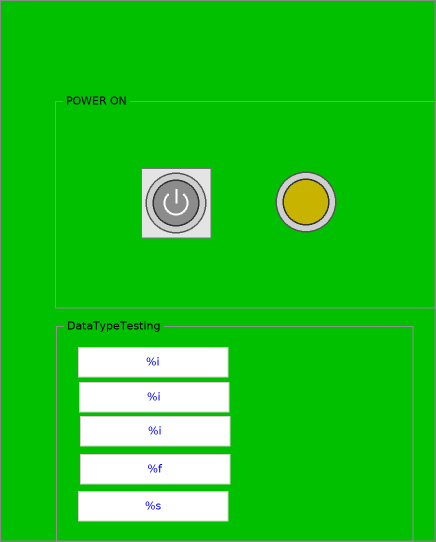
VISUALIZATION HMI  // 436x542
    GroupBox (55,93 381x215), "POWER ON"
        Lamp1 (216,74 70x70), variable: MAIN.bEnable, style: Lamp-Lamp1-Yellow
        PowerSwitch (86,75 70x70), variable: MAIN.bStart, behaviour: TOGGLE, style: Switch-PowerSwitch-Gray
    GroupBox (56,318 357x224), "DataTypeTesting"
        Textfield (22,29 150x30), "%i", text variable: MAIN.bEnable
        Textfield (23,64 150x30), "%i", text variable: MAIN.nINT
        Textfield (22,173 150x30), "%s", text variable: MAIN.sPowerStatus
            OnMouseDown: write the text variable via Default
        Textfield (24,136 150x30), "%f", text variable: MAIN.fREAL
            OnMouseDown: write the text variable via Default, min 0, max 1
        Textfield (24,98 150x30), "%i", text variable: MAIN.nUINT
END_VISUALIZATION

(* stored: Version 1.1.0.1, ProductVersion 3.1.4024.12
   Visu HMI: Id {005e27fe-70c2-482d-8f3f-557973bb7fb7} *)
